PROGRAM EM01_Dispenser
VAR
END_VAR

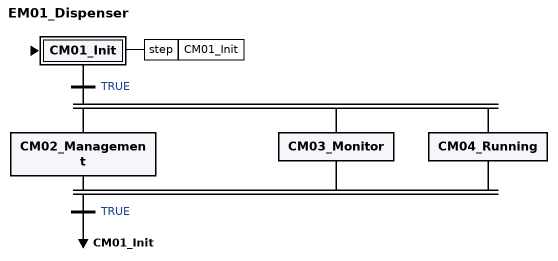
INITIAL_STEP CM01_Init:
    CM01_Init(N);  // step action
END_STEP
TRANSITION FROM CM01_Init TO (CM02_Management, CM03_Monitor, CM04_Running)
    := TRUE;
END_TRANSITION
STEP CM02_Management:
END_STEP
STEP CM03_Monitor:
END_STEP
STEP CM04_Running:
END_STEP
TRANSITION FROM (CM02_Management, CM03_Monitor, CM04_Running) TO CM01_Init
    := TRUE;
END_TRANSITION

ACTION CM01_Init:

END_ACTION

ACTION CM02_Management:
// NETWORK 1
END_ACTION

ACTION CM03_Monitor:
// NETWORK 1
END_ACTION

ACTION CM04_Running:
// NETWORK 1
END_ACTION

END_PROGRAM

(* stored: Version 1.1.0.1, ProductVersion 3.1.4024.9
   POU EM01_Dispenser: Id {4b5cbac8-95c4-4e6d-b826-0d0dce5f5a21}, SpecialFunc None
   Action CM01_Init: Id {2f3697b2-d968-4623-8b73-9504eb580f8b}
   Action CM02_Management: Id {23e9dfb0-aa7e-41a1-9d3a-f57463d513f4}
   Action CM03_Monitor: Id {15fa63c8-13b0-421f-9a16-dc294a9a5d46}
   Action CM04_Running: Id {12925d05-9a0c-4141-b521-429fef0d2ba0} *)
